{attribute 'GeneratedUsingTerminal: EK1122-0000-0018'}
{attribute addProperty BoxType "EK1122-0000-0018"}
{attribute addProperty Id "RC60_VI_AES_D_BC_ECAT_xAES_A3B0707168RC60_SAFETY_Flexi_Soft_EtherCAT_GatewayFlexi_Soft_EtherCAT_Gateway_DE394EDD5"}
{attribute addProperty CRC "1644325056"}
{attribute addProperty Size "73"}
{attribute addProperty Name "RC60_A2 (EK1122)"}
TYPE RC60_A2_EK1122_620268C0 EXTENDS EK1122_1FC0878B : 
STRUCT
    {attribute addProperty Name "RC60_VI (AES-D-BC-ECAT)"}
    {attribute addProperty PreviousPort "RC60_A2 (EK1122) : D"}
    {attribute addProperty SyncUnit "C60"}
    RC60_VI_AES_D_BC_ECAT_x : AES_A3B07071;
    {attribute addProperty Name "RC60_SAFETY (Flexi Soft EtherCAT Gateway)"}
    {attribute addProperty PreviousPort "RC60_A2 (EK1122) : B"}
    {attribute addProperty SyncUnit "C60"}
    RC60_SAFETY_Flexi_Soft_EtherCAT_Gateway : Flexi_Soft_EtherCAT_Gateway_DE394EDD;
END_STRUCT
END_TYPE

(* stored: Version 1.2.0.0, ProductVersion 3.1.4024.11
   DUT RC60_A2_EK1122_620268C0: Id {da9027bb-dbca-0ca8-381b-0e208d49ee14} *)
